KUKA KRL program: DEMO_PROC07.src, DEMO_PROC07.dat

--- DEMO_PROC07.src ---
&ACCESS RVO
&REL 4
&COMMENT Proc07
&PARAM DISKPATH = KRC:\R1\Program\PlcDemo
DEF  DEMO_PROC07 ( )
;********************************

;CREATOR : SPEEDBOT
;DATE    : 2024-09-23
;PROGRAM : DEMO_PROC07

;********************************
;FOLD INI;%{PE}
  ;FOLD BASISTECH INI
    GLOBAL INTERRUPT DECL 3 WHEN $STOPMESS==TRUE DO IR_STOPM ( )
    INTERRUPT ON 3
    BAS (#INITMOV,0 )
  ;ENDFOLD (BASISTECH INI)
  ;FOLD USER INI
    ;Make your modifications here
    continue
    if $MOVE_BCO == FALSE Then
      ; BCO
      ptp cur_jpos_()
    endif
  ;ENDFOLD (USER INI)
;ENDFOLD (INI)

;Example program for Process 1

;waiting for PLC clearance to proceed
;FOLD PLC.RequestToContinue ;%{PE}
req_to_continue_()
;ENDFOLD
;FOLD PLC.PathSegment IN Segment Nr: 126 ;%{PE}
path_segment_(126)
;ENDFOLD

;entering interference zone 1 with robot *.
;Enter Zone With R***
;FOLD PLC.EnterZone IN Zone Nr: ZONE [1] ;%{PE}
zone_ctrl_(#I_ENTER, 1)
;ENDFOLD

;Teach the robot the process trajectory
;FOLD SPTP P1 CONT Vel=100 % PDAT1 Tool[1] Base[0] ;%{PE}
;FOLD Parameters ;%{h}
;Params IlfProvider=kukaroboter.basistech.inlineforms.movement.spline; Kuka.IsGlobalPoint=False; Kuka.PointName=P1; Kuka.BlendingEnabled=True; Kuka.MoveDataPtpName=PDAT1; Kuka.VelocityPtp=100; Kuka.VelocityFieldEnabled=True; Kuka.ColDetectFieldEnabled=True; Kuka.CurrentCDSetIndex=0; Kuka.MovementParameterFieldEnabled=True; IlfCommand=SPTP
;ENDFOLD
SPTP XP1 WITH $VEL_AXIS[1] = SVEL_JOINT(100.0), $TOOL = STOOL2(FP1), $BASE = SBASE(FP1.BASE_NO), $IPO_MODE = SIPO_MODE(FP1.IPO_FRAME), $LOAD = SLOAD(FP1.TOOL_NO), $ACC_AXIS[1] = SACC_JOINT(PPDAT1), $APO = SAPO_PTP(PPDAT1), $GEAR_JERK[1] = SGEAR_JERK(PPDAT1), $COLLMON_TOL_PRO[1] = USE_CM_PRO_VALUES(0) C_Spl
;ENDFOLD
;FOLD SPTP P2 CONT Vel=100 % PDAT2 Tool[1] Base[0] ;%{PE}
;FOLD Parameters ;%{h}
;Params IlfProvider=kukaroboter.basistech.inlineforms.movement.spline; Kuka.IsGlobalPoint=False; Kuka.PointName=P2; Kuka.BlendingEnabled=True; Kuka.MoveDataPtpName=PDAT2; Kuka.VelocityPtp=100; Kuka.VelocityFieldEnabled=True; Kuka.ColDetectFieldEnabled=True; Kuka.CurrentCDSetIndex=0; Kuka.MovementParameterFieldEnabled=True; IlfCommand=SPTP
;ENDFOLD
SPTP XP2 WITH $VEL_AXIS[1] = SVEL_JOINT(100.0), $TOOL = STOOL2(FP2), $BASE = SBASE(FP2.BASE_NO), $IPO_MODE = SIPO_MODE(FP2.IPO_FRAME), $LOAD = SLOAD(FP2.TOOL_NO), $ACC_AXIS[1] = SACC_JOINT(PPDAT2), $APO = SAPO_PTP(PPDAT2), $GEAR_JERK[1] = SGEAR_JERK(PPDAT2), $COLLMON_TOL_PRO[1] = USE_CM_PRO_VALUES(0) C_Spl
;ENDFOLD
;FOLD SPTP P3 CONT Vel=100 % PDAT3 Tool[1] Base[0] ;%{PE}
;FOLD Parameters ;%{h}
;Params IlfProvider=kukaroboter.basistech.inlineforms.movement.spline; Kuka.IsGlobalPoint=False; Kuka.PointName=P3; Kuka.BlendingEnabled=True; Kuka.MoveDataPtpName=PDAT3; Kuka.VelocityPtp=100; Kuka.VelocityFieldEnabled=True; Kuka.ColDetectFieldEnabled=True; Kuka.CurrentCDSetIndex=0; Kuka.MovementParameterFieldEnabled=True; IlfCommand=SPTP
;ENDFOLD
SPTP XP3 WITH $VEL_AXIS[1] = SVEL_JOINT(100.0), $TOOL = STOOL2(FP3), $BASE = SBASE(FP3.BASE_NO), $IPO_MODE = SIPO_MODE(FP3.IPO_FRAME), $LOAD = SLOAD(FP3.TOOL_NO), $ACC_AXIS[1] = SACC_JOINT(PPDAT3), $APO = SAPO_PTP(PPDAT3), $GEAR_JERK[1] = SGEAR_JERK(PPDAT3), $COLLMON_TOL_PRO[1] = USE_CM_PRO_VALUES(0) C_Spl
;ENDFOLD


;This position has been fully cleared
;Does not interfere with the gripper and the corresponding robot.

;Report placement complete
;FOLD PLC.PathSegment IN Segment Nr: 156;%{PE}
path_segment_(156)
;ENDFOLD

;Exit the interference zone 1 with robot *.
;Enter Zone With R***
;FOLD PLC.ExitZone IN Zone Nr: ZONE [1] ;%{PE}
zone_ctrl_(#I_EXIT, 1)
;ENDFOLD
END

--- DEMO_PROC07.dat ---
&ACCESS RVO
&REL 4
&COMMENT Proc07
&PARAM DISKPATH = KRC:\R1\Program\PlcDemo
DEFDAT  DEMO_PROC07
;FOLD EXTERNAL DECLARATIONS;%{PE}%MKUKATPBASIS,%CEXT,%VCOMMON,%P
;FOLD BASISTECH EXT;%{PE}%MKUKATPBASIS,%CEXT,%VEXT,%P
EXT  BAS (BAS_COMMAND  :IN,REAL  :IN )
DECL INT SUCCESS
;ENDFOLD (BASISTECH EXT)
;FOLD USER EXT;%{E}%MKUKATPUSER,%CEXT,%VEXT,%P
;Make your modifications here

;ENDFOLD (USER EXT)
;ENDFOLD (EXTERNAL DECLARATIONS)
DECL E6POS XP1={X 0.00,Y 0.0,Z 0.00,A 0.0,B 0.0000,C 0.0,S 0,T 2,E1 0.0,E2 0.0,E3 0.0,E4 0.0,E5 0.0,E6 0.0}
DECL FDAT FP1={TOOL_NO 1,BASE_NO 0,IPO_FRAME #BASE,POINT2[] " "}
DECL PDAT PPDAT1={VEL 100.000,ACC 100.000,APO_DIST 500.000,APO_MODE #CDIS,GEAR_JERK 100.000,EXAX_IGN 0}
DECL MODULEPARAM_T LAST_TP_PARAMS={PARAMS[] "Kuka.VelocityFieldEnabled=True; Kuka.ColDetectFieldEnabled=True; Kuka.MovementParameterFieldEnabled=True; Kuka.IsAngleEnabled=False; Kuka.PointName=P3; Kuka.FrameData.base_no=0; Kuka.FrameData.tool_no=1; Kuka.FrameData.ipo_frame=#BASE; Kuka.isglobalpoint=False; Kuka.MoveDataPtpName=PDAT3; Kuka.MovementDataPdat.apo_mode=#CDIS; Kuka.MovementDataPdat.apo_dist=500; Kuka.MovementData.vel=100; Kuka.MovementData.acc=100; Kuka.MovementData.gear_jerk=100; Kuka.MovementData.exax_ign=0; Kuka.VelocityPtp=100; Kuka.BlendingEnabled=True; Kuka.CurrentCDSetIndex=0    "}
DECL E6POS XP2={X 0.00,Y 0.0,Z 0.00,A 0.0,B 0.0000,C 0.0,S 0,T 2,E1 0.0,E2 0.0,E3 0.0,E4 0.0,E5 0.0,E6 0.0}
DECL FDAT FP2={TOOL_NO 1,BASE_NO 0,IPO_FRAME #BASE,POINT2[] " "}
DECL PDAT PPDAT2={VEL 100.000,ACC 100.000,APO_DIST 500.000,APO_MODE #CDIS,GEAR_JERK 100.000,EXAX_IGN 0}
DECL E6POS XP3={X 0.00,Y 0.0,Z 0.00,A 0.0,B 0.0000,C 0.0,S 0,T 2,E1 0.0,E2 0.0,E3 0.0,E4 0.0,E5 0.0,E6 0.0}
DECL FDAT FP3={TOOL_NO 1,BASE_NO 0,IPO_FRAME #BASE,POINT2[] " "}
DECL PDAT PPDAT3={VEL 100.000,ACC 100.000,APO_DIST 500.000,APO_MODE #CDIS,GEAR_JERK 100.000,EXAX_IGN 0}
ENDDAT
